// Mitsubishi GX Works2 project: COUNTERS   PLC: Q02/Q02H

PROGRAM COUNT
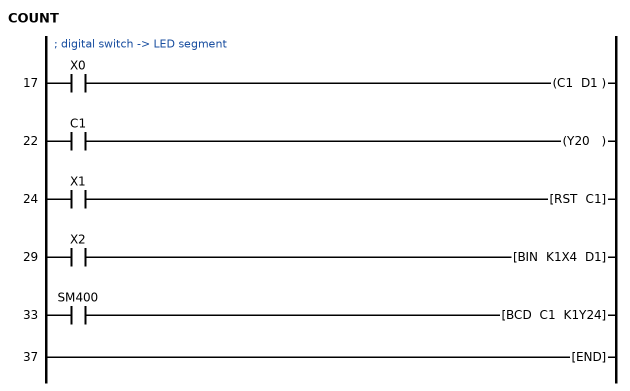
; digital switch -> LED segment
17    LD      X0
      OUT     C1 D1
22    LD      C1
      OUT     Y20
24    LD      X1
      RST     C1
29    LD      X2
      BIN     K1X4 D1
33    LD      SM400
      BCD     C1 K1Y24
37    END
END_PROGRAM
